// TIA Portal V17 export
// export: Created 2026-05-13T16:31:12.3845667Z, ExportSetting WithDefaults, DisplayName Totally Integrated Automation Portal, DisplayVersion V17 Update 4, DisplayName TIA Portal Openness, DisplayVersion V17 Update 4, DisplayName TIA Portal Version Control Interface, DisplayVersion V17, DisplayName SINAMICS Startdrive Advanced, DisplayVersion V17, DisplayName SINAMICS Startdrive G130, G150, S120, S150, SINAMICS MV, S210, DisplayVersion V17, DisplayName SINAMICS Startdrive G110M, G120, G120C, G120D, G120P, G115D, DisplayVersion V17, DisplayName STEP 7 Professional, DisplayVersion V17 Update 4, DisplayName STEP 7 Safety, DisplayVersion V17, DisplayName WinCC Professional, DisplayVersion V17 Update 4
TagTable "Codex_Popup_PLC_Named_Int_Tags"
  DB_Components_Valve01_ClickTrig : Bool  (PLC tag DB_Components.Valve01.ClickTrig, HMI_连接_1, 1 s, start 0)   // PLC linked: DB_Components.Valve01.ClickTrig.
  DB_Components_Valve01_DoubleClickTime : Int  (1 s, start 0)   // Internal helper only. DB_Components.Valve01 has no DoubleClickTime member in the exported PLC DB.
  DB_Components_Valve01_Switch1 : Bool  (PLC tag DB_Components.Valve01.Switch[1], HMI_连接_1, 1 s, start 0)   // PLC linked: DB_Components.Valve01.Switch[1].
  DB_Components_Valve01_RealValue1 : Real  (PLC tag DB_Components.Valve01.RealValue[1], HMI_连接_1, 1 s)   // PLC linked: DB_Components.Valve01.RealValue[1].
  DB_Components_Valve01_RealValue1_Int : Int  (1 s, start 0)   // Legacy Int placeholder kept for screens that still use the Int simulation field.
  DB_ActivePopup_Valve01_Visible : Bool  (PLC tag DB_ActivePopup.Valve01.Visible, HMI_连接_1, 1 s, start 0)   // PLC linked: DB_ActivePopup.Valve01.Visible.
  DB_ActivePopup_Valve01_ActiveID : Int  (PLC tag DB_ActivePopup.Valve01.ActiveID, HMI_连接_1, 1 s, start 0)   // PLC linked: DB_ActivePopup.Valve01.ActiveID.
  DB_ActivePopup_Valve01_Confirmed : Bool  (PLC tag DB_ActivePopup.Valve01.Confirmed, HMI_连接_1, 1 s, start 0)   // PLC linked: DB_ActivePopup.Valve01.Confirmed.
  DB_ActivePopup_Valve01_ConfirmBtn : Bool  (PLC tag DB_ActivePopup.Valve01.ConfirmBtn, HMI_连接_1, 1 s, start 0)   // PLC linked: DB_ActivePopup.Valve01.ConfirmBtn.
  DB_ActivePopup_Valve01_CancelBtn : Bool  (PLC tag DB_ActivePopup.Valve01.CancelBtn, HMI_连接_1, 1 s, start 0)   // PLC linked: DB_ActivePopup.Valve01.CancelBtn.
  DB_Components_Heater01_ClickTrig : Bool  (PLC tag DB_Components.Heater01.ClickTrig, HMI_连接_1, 1 s, start 0)   // PLC linked: DB_Components.Heater01.ClickTrig.
  DB_Components_Heater01_DoubleClickTime : Int  (1 s, start 0)   // Internal helper only. DB_Components.Heater01 has no DoubleClickTime member in the exported PLC DB.
  DB_Components_Heater01_Switch1 : Bool  (PLC tag DB_Components.Heater01.Switch[1], HMI_连接_1, 1 s, start 0)   // PLC linked: DB_Components.Heater01.Switch[1].
  DB_Components_Heater01_RealValue1 : Real  (PLC tag DB_Components.Heater01.RealValue[1], HMI_连接_1, 1 s)   // PLC linked: DB_Components.Heater01.RealValue[1].
  DB_Components_Heater01_RealValue1_Int : Int  (1 s, start 0)   // Legacy Int placeholder kept for screens that still use the Int simulation field.
  DB_ActivePopup_Heater01_Visible : Bool  (PLC tag DB_ActivePopup.Heater01.Visible, HMI_连接_1, 1 s, start 0)   // PLC linked: DB_ActivePopup.Heater01.Visible.
  DB_ActivePopup_Heater01_Confirmed : Bool  (PLC tag DB_ActivePopup.Heater01.Confirmed, HMI_连接_1, 1 s, start 0)   // PLC linked: DB_ActivePopup.Heater01.Confirmed.
  DB_ActivePopup_Heater01_ConfirmBtn : Bool  (PLC tag DB_ActivePopup.Heater01.ConfirmBtn, HMI_连接_1, 1 s, start 0)   // PLC linked: DB_ActivePopup.Heater01.ConfirmBtn.
  DB_ActivePopup_Heater01_CancelBtn : Bool  (PLC tag DB_ActivePopup.Heater01.CancelBtn, HMI_连接_1, 1 s, start 0)   // PLC linked: DB_ActivePopup.Heater01.CancelBtn.
  DB_Components_Fan01_ClickTrig : Bool  (PLC tag DB_Components.Fan01.ClickTrig, HMI_连接_1, 1 s, start 0)   // PLC linked: DB_Components.Fan01.ClickTrig.
  DB_Components_Fan01_DoubleClickTime : Int  (1 s, start 0)   // Internal helper only. DB_Components.Fan01 has no DoubleClickTime member in the exported PLC DB.
  DB_Components_Fan01_Switch1 : Bool  (PLC tag DB_Components.Fan01.Switch[1], HMI_连接_1, 1 s, start 0)   // PLC linked: DB_Components.Fan01.Switch[1].
  DB_Components_Fan01_RealValue1 : Real  (PLC tag DB_Components.Fan01.RealValue[1], HMI_连接_1, 1 s)   // PLC linked: DB_Components.Fan01.RealValue[1].
  DB_Components_Fan01_RealValue1_Int : Int  (1 s, start 0)   // Legacy Int placeholder kept for screens that still use the Int simulation field.
  DB_ActivePopup_Fan01_Visible : Bool  (PLC tag DB_ActivePopup.Fan01.Visible, HMI_连接_1, 1 s, start 0)   // PLC linked: DB_ActivePopup.Fan01.Visible.
  DB_ActivePopup_Fan01_ActiveID : Int  (PLC tag DB_ActivePopup.Fan01.ActiveID, HMI_连接_1, 1 s, start 0)   // PLC linked: DB_ActivePopup.Fan01.ActiveID.
  DB_ActivePopup_Fan01_Confirmed : Bool  (PLC tag DB_ActivePopup.Fan01.Confirmed, HMI_连接_1, 1 s, start 0)   // PLC linked: DB_ActivePopup.Fan01.Confirmed.
  DB_ActivePopup_Fan01_ConfirmBtn : Bool  (PLC tag DB_ActivePopup.Fan01.ConfirmBtn, HMI_连接_1, 1 s, start 0)   // PLC linked: DB_ActivePopup.Fan01.ConfirmBtn.
  DB_ActivePopup_Fan01_CancelBtn : Bool  (PLC tag DB_ActivePopup.Fan01.CancelBtn, HMI_连接_1, 1 s, start 0)   // PLC linked: DB_ActivePopup.Fan01.CancelBtn.
